FUNCTION_BLOCK STOPGO (* ECC with no Transient ECC State *)
  (* Standard: 61499-2 *)
  (* Version 0.0, 2018-12-17, JHC, Holobloc Inc *)
  (* Compiler header: package fb.rt.test; *)
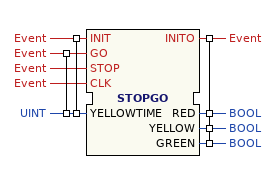
  EVENT_INPUT
    INIT WITH YELLOWTIME; (* Initialization Request *)
    GO WITH YELLOWTIME; (* Normal Execution Request *)
    STOP;
    CLK;
  END_EVENT
  EVENT_OUTPUT
    INITO WITH RED, YELLOW, GREEN; (* Initialization Confirm *)
  END_EVENT
  VAR_INPUT
    YELLOWTIME : UINT; (* Input event qualifier *)
  END_VAR
  VAR_OUTPUT
    RED : BOOL; (* Output event qualifier *)
    YELLOW : BOOL;
    GREEN : BOOL;
  END_VAR
  VAR
    YELLOWDONE : BOOL;
  END_VAR
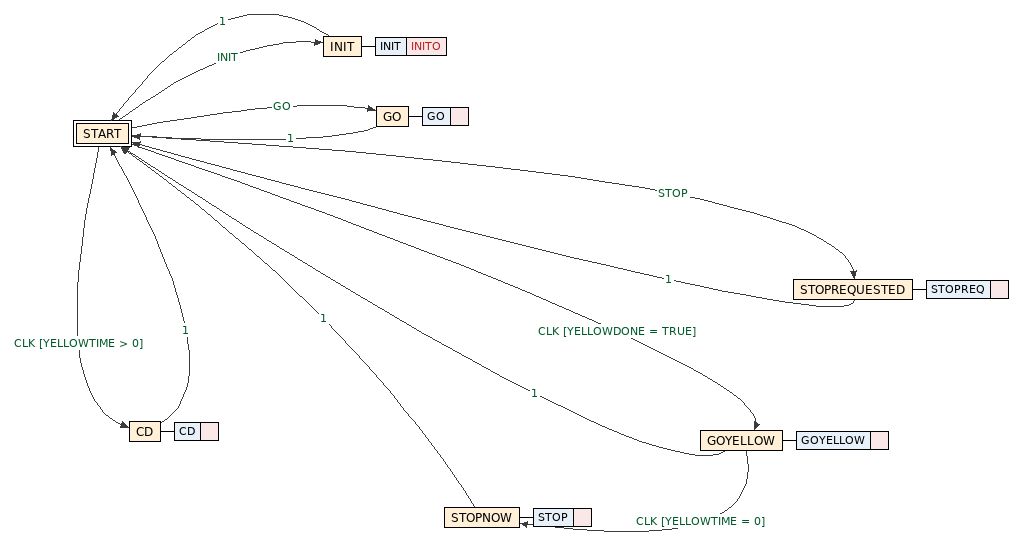
  EC_STATES
    START; (* Initial State *)
    INIT : INIT -> INITO; (* Initialization *)
    GO : GO;
    GOYELLOW : GOYELLOW;
    CD : CD;
    STOPNOW : STOP;
    STOPREQUESTED : STOPREQ;
  END_STATES
  EC_TRANSITIONS
    INIT TO START := 1;
    START TO INIT := INIT;
    START TO GO := GO;
    GO TO START := 1;
    START TO CD := CLK [YELLOWTIME > 0];
    GOYELLOW TO STOPNOW := CLK [YELLOWTIME = 0];
    STOPNOW TO START := 1;
    CD TO START := 1;
    START TO STOPREQUESTED := STOP;
    START TO GOYELLOW := CLK [YELLOWDONE = TRUE];
    GOYELLOW TO START := 1;
    STOPREQUESTED TO START := 1;
  END_TRANSITIONS
  ALGORITHM INIT IN ST: (* Initialization algorithm *)
RED:=FALSE;
YELLOW:=FALSE;
GREEN:=FALSE;
YELLOWDONE:=FALSE;
  END_ALGORITHM
  ALGORITHM STOP IN ST:
IF YELLOWTIME = 0 THEN
	RED:= TRUE;
	GREEN:= FALSE;
	YELLOW:= FALSE;
END_IF;
  END_ALGORITHM
  ALGORITHM GO IN ST:
GREEN:=TRUE;
YELLOW:=FALSE;
RED:=FALSE;
  END_ALGORITHM
  ALGORITHM CD IN ST:
YELLOWTIME:= YELLOWTIME - 1:
  END_ALGORITHM
  ALGORITHM GOYELLOW IN ST:
YELLOW:=TRUE;
RED:=FALSE;
GREEN:=FALSE;
  END_ALGORITHM
  ALGORITHM STOPREQ IN ST:

  END_ALGORITHM
END_FUNCTION_BLOCK
